Fanuc KAREL source: kt00890.KL

PROGRAM KT00890
%STACKSIZE=65535
%PRIORITY=65535
%NOLOCKGROUP
VAR
P1 : XYZWPREXT
P2 : XYZWPREXT
OUT : POSITION
BEGIN
P1.X=1.0
P2.Y=2.0
P1.X=1.0
P2.Y=2.0
-- UNRESOLVED_PC line 12 opcodes [27 27 49 7E AD 76 7E 4A] marker_code=80
END KT00890
